ABB RobotStudio station: Sesion5erronea.rspag

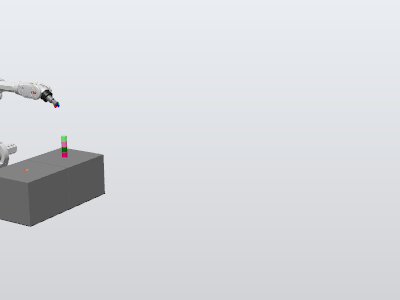
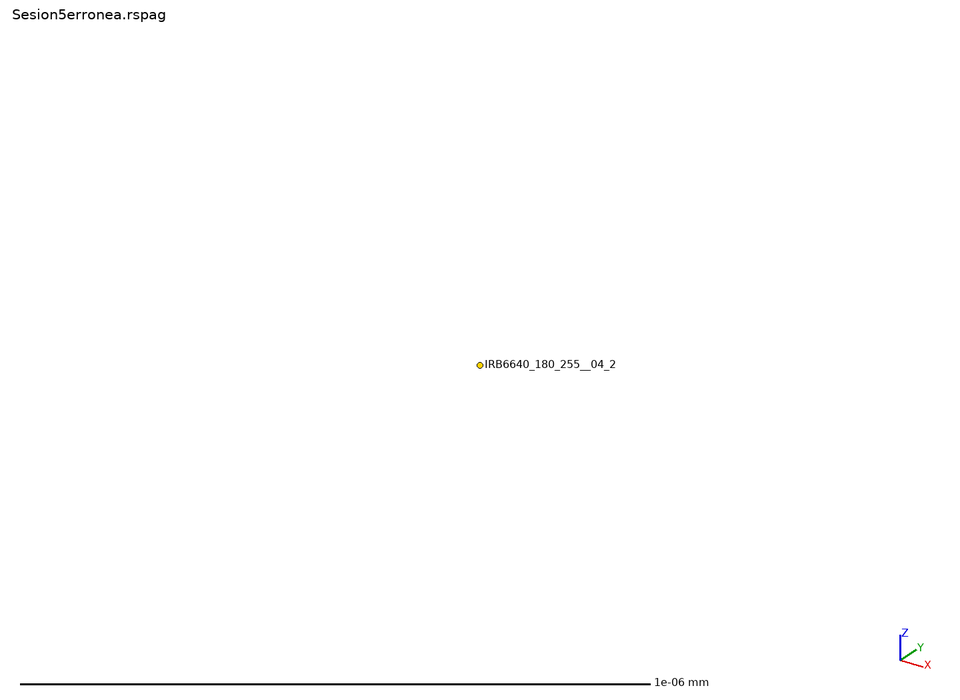
[picture v1: parts stored in the station drawn from their meshes, with robot base, taught points and paths (robot models come from the ABB library and are not in the file)]
--- station ---
Station Sesion3Prueba (saved by RobotStudio 24.1.10713.1)
Controller Controlador6
  mechanical unit ROB_1: IRB6640_180_255__04_2, 6 joints, base frame (0, 0, 0) mm
Layout (positions relative to the parent item):
  - Ventosa [mechanism] at (1635.71, 0, 1955) mm, rotated rx 180 ry 60 rz 180 deg
      TCP Ventosa at (0, 0, 200) mm
      links: PiezaVentosa
  - IRB6640_180_255__04_2 [mechanism, from %ABB.RobotStudio.Models.IRB6640%\IRB6640_180_255_G_04.rslib] at (0, 0, 0) mm; joint values [0, 0, 0, 0, 0.5236, 0] (rad or m)
  - MesaTrabajoParteIzq [part], size 1000 x 1000 x 750 mm
  - MesaTrabajoParteDer [part], size 1000 x 1000 x 750 mm
  - Componente inteligente_1 [smart component]
      signals: DO Vacuostato, DI ActivaVentosa
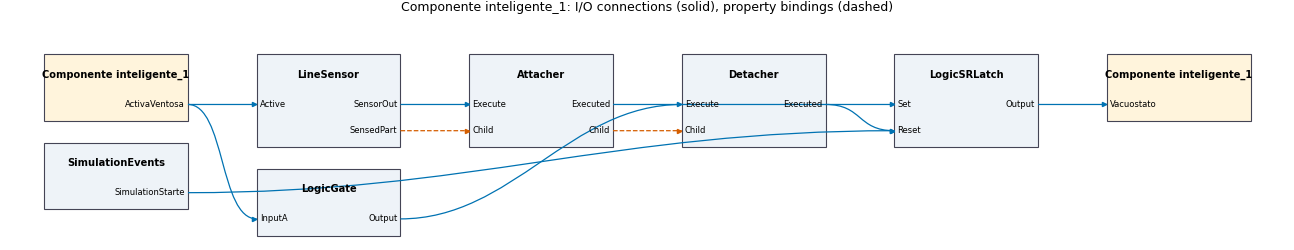
      connections:
        Componente inteligente_1.ActivaVentosa -> LineSensor.Active
        Componente inteligente_1.ActivaVentosa -> LogicGate.InputA
        LineSensor.SensorOut -> Attacher.Execute
        Attacher.Executed -> LogicSRLatch.Set
        LogicSRLatch.Output -> Componente inteligente_1.Vacuostato
        Detacher.Executed -> LogicSRLatch.Reset
        SimulationEvents.SimulationStarted -> LogicSRLatch.Reset
        LogicGate.Output -> Detacher.Execute
        LineSensor.SensedPart => Attacher.Child
        Attacher.Child => Detacher.Child
    - SimulationEvents [smart component, from Components\SimulationEvents.rslib]
    - LineSensor [smart component, from Components\LineSensor.rslib] at (1808.91, 0, 1855) mm, rotated rx 180 ry 60 rz 180 deg
        properties: Start=[0 0 -0.002]; End=[0 0 0.02]; Radius=0.002; SensedPart=Pieza_7; SensedPoint=[1.50000012207031 -0.500000030517578 0.85]; Length=0.022; Tag=(none)
      - _sensorPart_ [part], size 4 x 4 x 22 mm
    - LogicSRLatch [smart component, from Components\LogicSRLatch.rslib]
    - Attacher [smart component, from Components\Attacher.rslib]
        properties: Parent=Ventosa; Flange=0; Child=Pieza_7; Mount=false; Offset=[0 0 0]; Orientation=[0 0 0]
    - Detacher [smart component, from Components\Detacher.rslib]
        properties: Child=Pieza_7; KeepPosition=true
    - LogicGate [smart component, from Components\LogicGate.rslib]
        properties: Operator=NOT; Delay=0
  - Pieza_7 [part], size 100 x 99.8 x 100 mm
  - Pieza_9 [part] at (0, 0, 100) mm, size 100 x 99.8 x 100 mm
  - Pieza_10 [part] at (0, 0, 200) mm, size 100 x 99.8 x 100 mm
  - Pieza_11 [part] at (0, 0, 300) mm, size 100 x 99.8 x 100 mm
Attachment: Ventosa is attached to IRB6640_180_255__04_2 / Link6
Attachment: LineSensor is attached to Ventosa / PiezaVentosa
Station logic (signal -> signal, property => property):
  Controlador6.SD_ActivaVentosa -> Componente inteligente_1.ActivaVentosa
  Componente inteligente_1.Vacuostato -> Controlador6.ED_PiezaCogida

--- Backups/Controlador6/RAPID/TASK1/PROGMOD/CalibData.mod ---
MODULE CalibData
    PERS tooldata Ventosa:=[TRUE,[[0,0,200],[1,0,0,0]],[1,[0,0,125],[1,0,0,0],0,0,0.00125]];
ENDMODULE

--- Backups/Controlador6/RAPID/TASK1/PROGMOD/Module1.mod ---
MODULE Module1
    CONST robtarget pBaseTorre1:=[[1500,500,750],[0,0,1,0],[0,0,0,0],[9E+09,9E+09,9E+09,9E+09,9E+09,9E+09]];
    CONST robtarget pBaseTorre2:=[[1500,-500,750],[0,0,1,0],[-1,0,-1,0],[9E+09,9E+09,9E+09,9E+09,9E+09,9E+09]];
    CONST robtarget pReposo:=[[1808.910161514,0,1855],[0.5,0,0.866025404,0],[0,0,0,0],[9E+09,9E+09,9E+09,9E+09,9E+09,9E+09]];


    PROC main()
       VAR robtarget pbt:= pBaseTorre1;
       trasladaTorre pbt,100,100,4;
    ENDPROC
    PROC trasladaTorre(robtarget pBaseTorre,num ap, num dp,num np)
        VAR robtarget pIntermedia:= pBaseTorre;
        VAR robtarget pDestino:= pBaseTorre;
        pIntermedia.trans.y:=  pBaseTorre.trans.y - 3*dp;
        pDestino.trans.y:= pBaseTorre.trans.y + 3*dp;
        trasladaTorreAux pBaseTorre, pIntermedia,ap, dp,np;
        WaitTime 3;
        trasladaTorreAux pIntermedia,pDestino,ap, dp,np;
    ENDPROC
    PROC trasladaTorreAux(robtarget pBaseOrigen,robTarget pBaseDestino, num ap, num dp,num np)
        VAR num i;
        VAR robtarget pBOri;
        VAR robtarget PBDesti;
        FOR i FROM np TO 1 STEP -1 DO
            pBOri:= pBaseOrigen;
            !toco por la superficie superior del cilindro
            pBOri.trans.z:= pBaseOrigen.trans.z + (i)*ap;!es i o i-1?
            pBDesti:= pBaseDestino;
            !toco la superficie de la mesa
            pBDesti.trans.z:= pBaseDestino.trans.z + (np-i)*ap;
            muevePieza pBOri,pBDesti;

        ENDFOR
    ENDPROC
    PROC muevePieza(robtarget pOrigen,robTarget pDestino)
        VAR robtarget pOrigenAprox := pOrigen;
        VAR robtarget pDestinoAprox := pDestino;
        VAR num alturaAprox:= 150;
        pOrigenAprox.trans.z := pOrigen.trans.z + alturaAprox;
        pDestinoAprox.trans.z := pDestino.trans.z + alturaAprox;
        MoveJ pOrigenAprox,v2000,z100,Ventosa\WObj:=wobj0;
        MoveL pOrigen,v300,fine,Ventosa\WObj:=wobj0;
        SetDO SD_ActivaVentosa, 1;! se puede combinar con mode LDO
        WaitDI ED_PiezaCogida, 1;
        MoveL pOrigenAprox,v300,z0,Ventosa\WObj:=wobj0;
        MoveJ pDestinoAprox,v2000,z100,Ventosa\WObj:=wobj0;
        MoveL pDestino,v300,fine,Ventosa\WObj:=wobj0;
        SetDO SD_ActivaVentosa, 0;
        WaitDI ED_PiezaCogida, 0;
        MoveL pDestinoAprox,v300,z0,Ventosa\WObj:=wobj0;
    ENDPROC


ENDMODULE

--- Backups/Controlador6/SYSPAR/EIO.cfg ---
EIO:CFG_1.0:6:1::
#
INDUSTRIAL_NETWORK:

      -Name "DeviceNet" -Label "DeviceNet Master/Slave Network" -Address "2"
#
DEVICENET_DEVICE:

      -Name "MiDeviceNet" -Label "MiDeviceNet"
#
DEVICENET_INTERNAL_DEVICE:

      -Name "DN_Internal_Device" -VendorName "ABB Robotics"\
      -ProductName "DeviceNet Internal Slave Device"
#
EIO_SIGNAL:

      -Name "ED_PiezaCogida" -SignalType "DI" -Device "MiDeviceNet"\
      -Label "ED_PiezaCogida" -DeviceMap "0" -Access "All"

      -Name "SD_ActivaVentosa" -SignalType "DO" -Device "MiDeviceNet"\
      -Label "SD_ActivaVentosa" -DeviceMap "0" -Access "All"
